# EPICS autosave request: opticsApp/Db/2slit_soft_settings.req
$(P)$(SLIT)xn.TWV
$(P)$(SLIT)xp.TWV
$(P)$(SLIT)size.TWV
$(P)$(SLIT)center.TWV
$(P)$(SLIT)xp.MRES
$(P)$(SLIT)xn.MRES
$(P)$(SLIT)size.MRES
$(P)$(SLIT)center.MRES
$(P)$(SLIT)xp.DESC
$(P)$(SLIT)xn.DESC
$(P)$(SLIT)size.DESC
$(P)$(SLIT)center.DESC
$(P)$(SLIT)xp.EGU
$(P)$(SLIT)xn.EGU
$(P)$(SLIT)size.EGU
$(P)$(SLIT)center.EGU
